// TIA Portal V18 export
VAR_GLOBAL   // PLC tag table "04_6 Costanti Nomi Attuatore Stz06"
END_VAR
VAR_GLOBAL CONSTANT   // user constants
   H601 : Int := 1;   // EV Apri/chiudi cesoia giunzione
END_VAR
